(* CODESYS project PackagingOfCubes_part2.project

Project tree, tasks and I/O mapping:
  Device : CODESYS Control Win V3, 3S - Smart Software Solutions GmbH, version 3.5.17.10
    application Application
      libraries: Standard, * (System); Util, * (System)
      task MainTask (cyclic, interval 10 ms, priority 1) calls PLC_PRG, Model
      program Model [ST]: MoveConveyorsACT, MoveBlueBoxACT, MoveGreenBoxACT, ChangeBoxACT, BoxSensorsACT, CheckFullACT
      image pool ImagePool
      visualisation Visualization
      data type SmallBox
      data type WoodenBox
      program PLC_PRG [SFC]: Alustus_active, Pakkaus_active, Vaihto_active
      global variables GVL
      function block HihnanOhjaus [FBD]
      program UnitTest [ST]
      visualisation Yksikkotestaus
  5ce3da45-db07-42e7-a21c-a00fff4ed8f6|C:\Users\Andrei\Downloads\crate-1143427_640.png
  text list GlobalTextList
*)

// Device/Application/SmallBox
TYPE SmallBox :
STRUCT
	x :REAL;
	sx :REAL;
	y :REAL;
	sy :REAL;
	rot :REAL;
END_STRUCT
END_TYPE

// Device/Application/WoodenBox
TYPE WoodenBox :
STRUCT
	scale :REAL := 1000.0;
	x :REAL;
	y :REAL;
	invisible :BOOL := TRUE;
END_STRUCT
END_TYPE

// Device/Application/GVL
VAR_GLOBAL
	// Sensors:
	sensorGreen : BOOL;
	sensorBlue : BOOL;
	boxNotFull : BOOL;
	
	// Actuators:
	startGreen : BOOL;
	startBlue : BOOL;
	changeBox : BOOL;
	pauseGreen : BOOL;
	pauseBlue : BOOL;
END_VAR

// Device/Application/PLC_PRG
PROGRAM PLC_PRG
VAR
	sinHihna:HihnanOhjaus;
	vihrHihna:HihnanOhjaus;
END_VAR

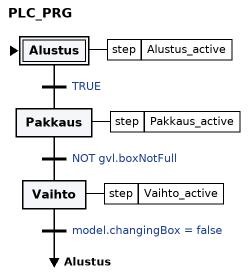
INITIAL_STEP Alustus:
    Alustus_active(N);  // step action
END_STEP
TRANSITION FROM Alustus TO Pakkaus
    := TRUE;
END_TRANSITION
STEP Pakkaus:
    Pakkaus_active(N);  // step action
END_STEP
TRANSITION FROM Pakkaus TO Vaihto
    := NOT gvl.boxNotFull;
END_TRANSITION
STEP Vaihto:
    Vaihto_active(N);  // step action
END_STEP
TRANSITION FROM Vaihto TO Alustus
    := model.changingBox = false;
END_TRANSITION

ACTION Alustus_active:
gvl.changeBox := FALSE;

vihrHihna.N := 3;
vihrHihna.restart := TRUE;

sinHihna.N := 5;
sinHihna.restart := TRUE;

vihrHihna.pause := gvl.pauseGreen;
sinHihna.pause := gvl.pauseBlue;
END_ACTION

ACTION Pakkaus_active:
vihrHihna();
sinHihna();
vihrHihna.restart := FALSE;
sinHihna.restart := FALSE;
vihrHihna.pause := gvl.pauseGreen;
sinHihna.pause := gvl.pauseBlue;
gvl.startGreen := vihrHihna.belt;
gvl.startBlue := sinHihna.belt;
vihrHihna.sensor := gvl.sensorGreen;
sinHihna.sensor := gvl.sensorBlue;
END_ACTION

ACTION Vaihto_active:
gvl.changeBox := TRUE;
gvl.startBlue := FALSE;
gvl.startGreen := FALSE;
END_ACTION

END_PROGRAM

// Device/Application/HihnanOhjaus
FUNCTION_BLOCK HihnanOhjaus
VAR_INPUT
	sensor:BOOL;
	restart:BOOL;
	N:INT;
	pause:BOOL;
END_VAR
VAR_OUTPUT
	belt:BOOL := TRUE;
	count:INT := 0;
END_VAR
VAR
	yksi_boxi: CTD;
END_VAR
VAR // added by the converter: edge detectors and wires of the graphical bodies
    _rt1 : R_TRIG;
END_VAR

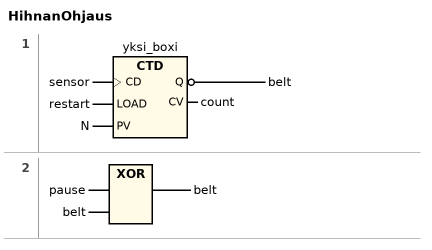
// NETWORK 1
_rt1(CLK := sensor);
yksi_boxi(CD := _rt1.Q, LOAD := restart, PV := N, CV => count); // CTD
belt := NOT yksi_boxi.Q;

// NETWORK 2
belt := pause XOR belt;

END_FUNCTION_BLOCK

// Device/Application/Model
PROGRAM Model
VAR
	// Define following variables according to needs
	blueBoxReq :INT := 5;
	greenBoxReq :INT := 3;
	maxSpeedBlueConv :REAL := 1.0;
	accBlueConv :REAL := 0.5;
	desaccBlueConv :REAL := 1.0;
	maxSpeedGreenConv :REAL := 1.17;
	accGreenConv :REAL := 0.5;
	desaccGreenConv :REAL := 1.0;
	gravityAcc :REAL := 8.0;
	cycleTime :REAL := 10;
END_VAR

VAR
	// Outputs from the model:
	blueSensor :BOOL;
	greenSensor :BOOL;
	boxNotFull :BOOL := TRUE;
	//////////////////////////
	// Inputs to the model:
	goBlueBelt :BOOL;	// Start the conveyor with blue boxes.
	goGreenBelt :BOOL;	// Start the conveyor with green boxes.
	changeBox :BOOL;	// Get a new wooden box.
	/////////////////////////
	nrBox :INT := 1;
	reqChangeBox :BOOL;
	blueBox :SmallBox;
	greenBox :SmallBox;
	speedBlueConv :REAL := 0.0;
	speedGreenConv :REAL := 0.0;
	rotAccBlueBox :REAL := 0.0;
	rotAccGreenBox :REAL := 0.0;
	blueInBox :INT := 0;
	greenInBox :INT := 0;
	posBlueConveyor :REAL := 0.0;
	posGreenConveyor :REAL := 0.0;
	blueBounced :BOOL;
	greenBounced :BOOL;
	woodBox1 :WoodenBox;
	changingBox :BOOL;
	wastedBoxes :INT;
END_VAR

// Read the inputs to the model, which correspond to the outputs from the controller:
goBlueBelt := GVL.startBlue;
goGreenBelt := GVL.startGreen;
changeBox := GVL.changeBox;

// Move conveyors as requested:
MoveConveyorsACT();

// Change wooden box if requested:
ChangeBoxACT();

// Implementation for the movement of the blue and green boxes. In practice, there
// is only one blue and one green box, which alternate locations (change invisible
// to the user).
// First blue box:
MoveBlueBoxACT();
// Second, green box:
MoveGreenBoxACT();

// Read Sensors:
BoxSensorsACT();

// Check if box is full:
CheckFullACT();

// Update outputs from the model:
GVL.sensorBlue := blueSensor;
GVL.sensorGreen := greenSensor;
GVL.boxNotFull := boxNotFull;

ACTION MoveConveyorsACT:
// Implementation of the movement of the belts. Two operations are used: one for
// accelerating the conveyor and another for stopping the conveyor.
IF goBlueBelt THEN
	IF (speedBlueConv + accBlueConv*cycleTime/1000) < maxSpeedBlueConv THEN
		speedBlueConv := speedBlueConv + desaccBlueConv*cycleTime/1000;
	ELSE
		speedBlueConv := maxSpeedBlueConv;
	END_IF
ELSE
	IF (speedBlueConv - desaccBlueConv*cycleTime/1000) > 0.0 THEN
		speedBlueConv := speedBlueConv - desaccBlueConv*cycleTime/1000;
	ELSE
		speedBlueConv := 0.0;
	END_IF
END_IF

IF goGreenBelt THEN
	IF ABS((speedGreenConv - accGreenConv*cycleTime/1000)) < maxSpeedGreenConv THEN
		speedGreenConv := speedGreenConv - desaccGreenConv*cycleTime/1000;
	ELSE
		speedGreenConv := - maxSpeedGreenConv;
	END_IF
ELSE
	IF (speedGreenConv + desaccGreenConv*cycleTime/1000) < 0.0 THEN
		speedGreenConv := speedGreenConv + desaccGreenConv*cycleTime/1000;
	ELSE
		speedGreenConv := 0.0;
	END_IF
END_IF

// Used for visualization of the conveyor movement
posBlueConveyor := posBlueConveyor + speedBlueConv;
IF posBlueConveyor > 12 THEN
	posBlueConveyor := 0.0;
END_IF

posGreenConveyor := posGreenConveyor + speedGreenConv;
IF posGreenConveyor < -12 THEN
	posGreenConveyor := 0.0;
END_IF
END_ACTION

ACTION MoveBlueBoxACT:
// Follow: if the box is on the conveyor, the box follows the movement of the conveyor belt
// (takes its speed)
IF (blueBox.x > -1) AND (blueBox.x < 208) AND (blueBox.y > -1) THEN
	blueBox.sx := speedBlueConv;
END_IF

// Once the middle of the box reaches the edge of the conveyor, its horizontal speed 
// is influenced by its falling speed while in touch with the conveyor.
IF (blueBox.x >= 208) AND (blueBox.x <= 225) THEN
	blueBox.sx := blueBox.sx + gravityAcc * cycleTime / 1000;
END_IF

// Change position of the box according to its speed.
blueBox.x := blueBox.x + blueBox.sx;

// Once the ball reaches more than half its side off the conveyor, it starts to fall
// and rotate until the "bottom" of the wooden box if the box is not full yet, or it
// follows a predefined path outside the box if its full.
// Box is over the edge, hence it starts to fall:
IF (blueBox.x >= 208) THEN
	blueBox.sy := blueBox.sy + gravityAcc * cycleTime / 1000;
END_IF

// Add the vertical speed to the position:
blueBox.y := blueBox.y + blueBox.sy;

// Rotation of the box: first calculate angular acceleration
IF (blueBox.x >= 208) AND (blueBox.x < 225) THEN
	rotAccBlueBox := COS(blueBox.sy / 17.0) + ATAN(gravityAcc / (blueBox.sx));
END_IF

// Then apply rotation:
blueBox.rot := blueBox.rot + rotAccBlueBox;

// IF wooden box is not full, return blue box to origin.
IF (blueInBox < blueBoxReq) AND (blueBox.y > 200) AND NOT(changingBox) THEN
	blueBox.x := 0.0;
	blueBox.y := 0.0;
	blueBox.rot := 0.0;
	blueBox.sy := 0.0;
	rotAccBlueBox := 0.0;
	blueInBox := blueInBox + 1;
END_IF

// If wooden box is full with blue boxes or being changed, box boinces out of wooden box
// Also, the wasted boxes counter is incremented
IF ((blueInBox >= blueBoxReq) OR changingBox) AND (blueBox.y > 110) AND NOT(blueBounced) THEN
	blueBox.sy := - blueBox.sy * 0.75;
	blueBounced := TRUE;
	wastedBoxes := wastedBoxes + 1;
END_IF
// Once it reaches some level, it returns to origin
IF (blueBox.y > 345) THEN
	blueBox.x := 0.0;
	blueBox.y := 0.0;
	blueBox.rot := 0.0;
	blueBox.sy := 0.0;
	rotAccBlueBox := 0.0;
	blueBounced := FALSE;
END_IF
END_ACTION

ACTION MoveGreenBoxACT:
// Follow: if the box is on the conveyor, the box follows the movement of the conveyor belt
// (takes its speed)
IF (greenBox.x < 1) AND (greenBox.x > -213) AND (greenBox.y > -1) THEN
	greenBox.sx := speedGreenConv;
END_IF

// Once the middle of the box reaches the edge of the conveyor, its horizontal speed 
// is influenced by its falling speed while in touch with the conveyor.
IF (greenBox.x <= -213) AND (greenBox.x >= -230) THEN
	greenBox.sx := greenBox.sx - gravityAcc * cycleTime / 1000;
END_IF

// Change position of the box according to its speed.
greenBox.x := greenBox.x + greenBox.sx;

// Once the ball reaches more than half its side off the conveyor, it starts to fall
// and rotate until the "bottom" of the wooden box if the box is not full yet, or it
// follows a predefined path outside the box if its full.
// Box is over the edge, hence it starts to fall:
IF (greenBox.x <= -213) THEN
	greenBox.sy := greenBox.sy + gravityAcc * cycleTime / 1000;
END_IF

// Add the vertical speed to the position:
greenBox.y := greenBox.y + greenBox.sy;

// Rotation of the box: first calculate angular acceleration
IF (greenBox.x <= -213) AND (greenBox.x >= -230) THEN
	rotAccGreenBox := ATAN(gravityAcc / greenBox.sx) - COS(blueBox.sy / 17.0);
END_IF

// Then apply rotation:
greenBox.rot := greenBox.rot + rotAccGreenBox;

// IF wooden box is not full or being changed, return blue box to origin.
IF (greenInBox < greenBoxReq) AND (greenBox.y > 200) AND NOT(changingBox) THEN
	greenBox.x := 0.0;
	greenBox.y := 0.0;
	greenBox.rot := 0.0;
	greenBox.sy := 0.0;
	rotAccGreenBox := 0.0;
	greenInBox := greenInBox + 1;
END_IF

// If wooden box is full with green boxes or being changed, box boinces out of wooden box
// Also, the wasted boxes counter is incremented
IF ((greenInBox >= greenBoxReq) OR changingBox) AND (greenBox.y > 110) AND NOT(greenBounced) THEN
	greenBox.sy := - greenBox.sy * 0.75;
	greenBounced := TRUE;
	wastedBoxes := wastedBoxes + 1;
END_IF
// Once it reaches some level, it returns to origin
IF (greenBox.y > 345) THEN
	greenBox.x := 0.0;
	greenBox.y := 0.0;
	greenBox.rot := 0.0;
	greenBox.sy := 0.0;
	rotAccGreenBox := 0.0;
	greenBounced := FALSE;
END_IF
END_ACTION

ACTION ChangeBoxACT:
// Edge detection mechanism: change the wooden box only on rising edge
IF changeBox AND NOT(reqChangeBox)THEN
	changingBox := TRUE;
	Model.woodBox1.invisible := FALSE;
	reqChangeBox := TRUE;
END_IF
IF NOT(changeBox) THEN
	reqChangeBox := FALSE;
END_IF

// Animation while the box is being changed
IF changingBox THEN
	IF (Model.woodBox1.y > -116) THEN
		Model.woodBox1.y := Model.woodBox1.y - 29 * cycleTime / 1000;
	ELSE
		Model.woodBox1.y := -116;
	END_IF
	IF (Model.woodBox1.scale > 600) THEN
		Model.woodBox1.scale := Model.woodBox1.scale - 100 * cycleTime / 1000;
	ELSE
		Model.woodBox1.scale := 600;
	END_IF
END_IF

// Once animation is done, return bozes to their original places and restore default values
IF changingBox AND (Model.woodBox1.y <= -116) AND (Model.woodBox1.scale <= 600) THEN
	Model.woodBox1.invisible := TRUE;
	Model.woodBox1.y := 0.0;
	Model.woodBox1.x := 0.0;
	Model.woodBox1.scale := 1000.0;
	nrBox := nrBox + 1;
	blueInBox := 0;
	greenInBox := 0;
	changingBox := FALSE;
END_IF
END_ACTION

ACTION BoxSensorsACT:
// Sensor to detect blue box
IF (blueBox.x > 213) AND (blueBox.x < 248) AND (blueBox.y < 20) THEN
	blueSensor := TRUE;
ELSE
	blueSensor := FALSE;
END_IF

IF (greenBox.x < -218) AND (greenBox.x > -253) AND (greenBox.y < 20) THEN
	greenSensor := TRUE;
ELSE
	greenSensor := FALSE;
END_IF
END_ACTION

ACTION CheckFullACT:
// Check if wooden box has both colours full or is being changed
IF ((blueInBox = blueBoxReq) AND (greenInBox = greenBoxReq)) OR changingBox THEN
	boxNotFull := FALSE;
ELSE
	boxNotFull := TRUE;
END_IF
END_ACTION

END_PROGRAM

// Device/Application/UnitTest
PROGRAM UnitTest
VAR
	hihna:HihnanOhjaus;
END_VAR

hihna.N := 5;
hihna();

END_PROGRAM

// Device/Application/Visualization
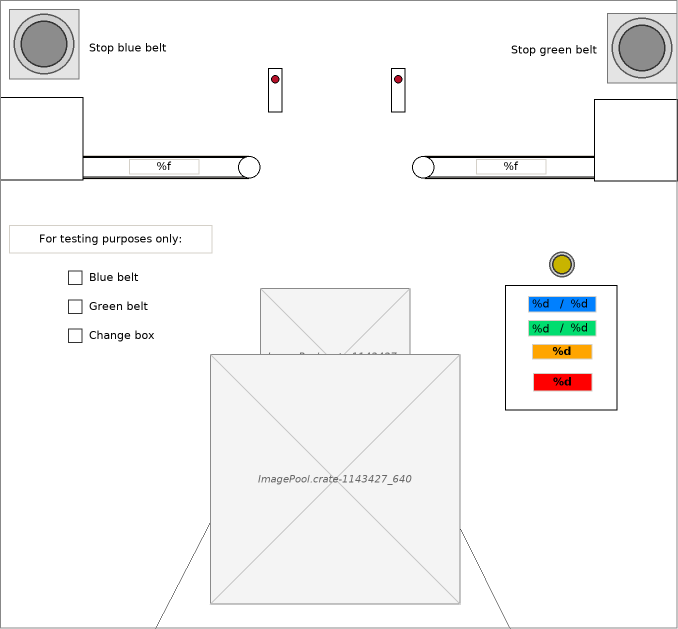
VISUALIZATION Visualization  // 678x629
    Rectangle (422,155 186x24)
    Rectangle (74,155 186x24)
    Line (71,178) (277,178)
        p3560616238: - Model.posBlueConveyor
    Line (51,156) (249,156)
        p3560616238: Model.posBlueConveyor
    Line (425,178) (602,178)
        p3560616238: - Model.posGreenConveyor
    Line (424,156) (601,156)
        p3560616238: Model.posGreenConveyor
    Rectangle (249,150 175x32)
    Rectangle (0,157 250x20)
    Rectangle (426,157 222x20)
    Polygon (155,629) (312,325) (360,326) (510,629)
    RoundedRectangle (505,285 112x125)
    Textfield (528,296 68x16), "/ %d", tooltip "Blue boxes packed", text variable: Model.blueBoxReq
    Textfield (527,297 28x14), "%d", text variable: Model.blueInBox
    Textfield (528,320 68x16), "/ %d", tooltip "Green boxes packed", text variable: Model.greenBoxReq
    Textfield (527,322 28x14), "%d", text variable: Model.greenInBox
    Ellipse (238,156 22x22)
    Ellipse (412,156 22x22)
    Checkbox (66,263 121x29), "Blue belt", variable: GVL.startBlue
    Checkbox (66,292 121x29), "Green belt", variable: GVL.startGreen
    Checkbox (66,321 121x29), "Change box", variable: GVL.changeBox
    Rectangle (25,120 35x35)
        p3560616238: Model.blueBox.x
        p2738717112: Model.blueBox.y
        p2858320360: Model.blueBox.rot
    Rectangle (620,120 35x35)
        p3560616238: Model.greenBox.x
        p2738717112: Model.greenBox.y
        p2858320360: Model.greenBox.rot
    Textfield (129,159 70x15), "%f", tooltip "Speed of conveyor", text variable: Model.speedBlueConv
    Textfield (476,159 70x15), "%f", tooltip "Speed of conveyor", text variable: Model.speedGreenConv
    Rectangle (268,68 14x44), tooltip "Blue boxes sensor"
    Ellipse (271,75 8x8)
    Ellipse (271,75 8x8), invisible if: Model.blueSensor
    Rectangle (391,68 14x44), tooltip "Green boxes sensor"
    Ellipse (394,75 8x8)
    Ellipse (394,75 8x8), invisible if: Model.greenSensor
    Lamp1 (547,249 30x31), tooltip "NotFull / Box in position", variable: Model.boxNotFull, style: Lamp-Lamp1-Yellow
    Image (260,288 150x150), image: ImagePool.crate-1143427_640
        p1097714728: Model.woodBox1.scale
    Rectangle (594,99 84x82)
    Rectangle (0,97 83x83)
    Image (210,354 250x250), image: ImagePool.crate-1143427_640
        p1097714728: Model.woodBox1.scale
        p3560616238: Model.woodBox1.x
        p2738717112: Model.woodBox1.y
    Textfield (532,344 60x15), "%d", tooltip "Box number", text variable: Model.nrBox
    Textfield (9,225 203x28), "For testing purposes only:"
    Textfield (533,373 59x18), "%d", tooltip "Wasted boxes", text variable: Model.wastedBoxes
    PushSwitch (607,13 70x70), variable: pauseGreen, behaviour: TOGGLE, style: Switch-PushSwitch-Gray
    PushSwitch (9,9 70x70), variable: pauseBlue, behaviour: TOGGLE, style: Switch-PushSwitch-Gray
    Label (479,35 150x30), "Stop green belt"
    Label (53,33 150x30), "Stop blue belt"
END_VISUALIZATION

// Device/Application/Yksikkotestaus
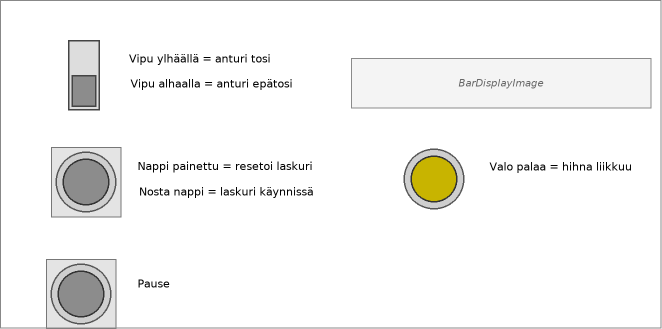
VISUALIZATION Yksikkotestaus  // 662x329
    Label (125,44 150x30), "Vipu ylhäällä = anturi tosi"
    BarDisplayImage (351,58 300x50), value: UnitTest.hihna.count, style: BarDisplayImage-Gray, scale format: %.1f, scale 0..5
    Lamp1 (399,144 70x70), variable: UnitTest.hihna.belt, style: Lamp-Lamp1-Yellow
    DipSwitch (49,40 70x70), variable: UnitTest.hihna.sensor, behaviour: TOGGLE, style: Switch-DipSwitch-Gray
    PushSwitch (51,147 70x70), variable: UnitTest.hihna.restart, behaviour: TOGGLE, style: Switch-PushSwitch-Gray
    Label (127,151 196x31), "Nappi painettu = resetoi laskuri"
    Label (133,177 187x30), "Nosta nappi = laskuri käynnissä"
    Label (460,152 202x30), "Valo palaa = hihna liikkuu"
    Label (122,69 179x30), "Vipu alhaalla = anturi epätosi"
    PushSwitch (46,259 70x70), variable: UnitTest.hihna.pause, behaviour: TOGGLE, style: Switch-PushSwitch-Gray
    Label (79,269 150x30), "Pause"
END_VISUALIZATION
